// TIA Portal V20 export
FUNCTION_BLOCK "FB - TableCheck"   // FB3, LAD
TITLE = Equipment - TableCheck
{ S7_Optimized_Access := 'TRUE' }
// This function block contains all logic for controlling a TableCheck module.
// -This module consists of a table, a jig presense sensor and Indication lamp Red (NG) and green (Ok).
// 
// >> Block created by: Engr. Awais Ali
// >> Block creation date:  08-10-2025
// stored: MemoryReserve 100, SetENOAutomatically false
   VAR_INPUT
      i_xJigPresent : Bool;
   END_VAR
   VAR_OUTPUT
      q_xLampNG : Bool;
      q_xLampOK : Bool;
   END_VAR
   VAR_IN_OUT
      iq_tableCheck : "UDT-TableCheck";
      iq_Sabload_L : "UDT-SABload";
      iq_Sabload_R : "UDT-SABload";
      iq_Bas342 : "UDT-BAS342";
   END_VAR
   VAR
      iState : Int;
      OnDelay_JigL { S7_SetPoint := 'True'} : TON_TIME;
      OffDelay_JigL { S7_SetPoint := 'True'} : TOF_TIME;
      OnDelay_JigR { S7_SetPoint := 'True'} : TON_TIME;
      OffDelay_JigR { S7_SetPoint := 'True'} : TOF_TIME;
   END_VAR
BEGIN

REGION Network 1: control - left jig
   // Detect the presence of left side Jig.
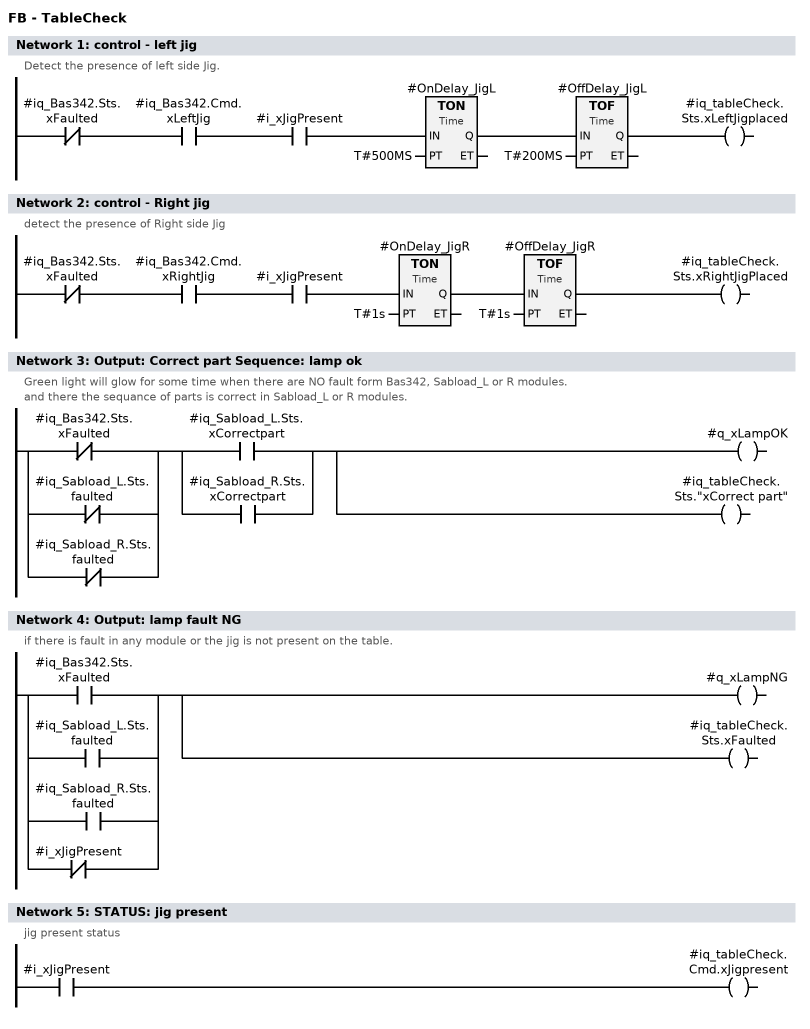
   RUNG wire#powerrail
      I_Contact( #iq_Bas342.Sts.xFaulted )
      Contact( #iq_Bas342.Cmd.xLeftJig )
      Contact( #i_xJigPresent )
      { S7_Templates := "time_type := Time" } #OnDelay_JigL.TON(pt := T#500MS, et =>)
      { S7_Templates := "time_type := Time" } #OffDelay_JigL.TOF(pt := T#200MS, et =>)
      Coil( #iq_tableCheck.Sts.xLeftJigplaced )
   END_RUNG
   // the same network as SCL:
   #OnDelay_JigL(IN := NOT #iq_Bas342.Sts.xFaulted AND #iq_Bas342.Cmd.xLeftJig AND #i_xJigPresent,   // TON
                 PT := T#500MS);
   #OffDelay_JigL(IN := #OnDelay_JigL.Q, PT := T#200MS);   // TOF
   #iq_tableCheck.Sts.xLeftJigplaced := #OffDelay_JigL.Q;
END_REGION

REGION Network 2: control - Right jig
   // detect the presence of Right side Jig
   RUNG wire#powerrail
      I_Contact( #iq_Bas342.Sts.xFaulted )
      Contact( #iq_Bas342.Cmd.xRightJig )
      Contact( #i_xJigPresent )
      { S7_Templates := "time_type := Time" } #OnDelay_JigR.TON(pt := T#1s, et =>)
      { S7_Templates := "time_type := Time" } #OffDelay_JigR.TOF(pt := T#1s, et =>)
      Coil( #iq_tableCheck.Sts.xRightJigPlaced )
   END_RUNG
   // the same network as SCL:
   #OnDelay_JigR(IN := NOT #iq_Bas342.Sts.xFaulted AND #iq_Bas342.Cmd.xRightJig AND #i_xJigPresent, PT := T#1s);   // TON
   #OffDelay_JigR(IN := #OnDelay_JigR.Q, PT := T#1s);   // TOF
   #iq_tableCheck.Sts.xRightJigPlaced := #OffDelay_JigR.Q;
END_REGION

REGION Network 3: Output: Correct part Sequence: lamp ok
   // Green light will glow for some time when there are NO fault form Bas342, Sabload_L or R modules. 
   // 
   // and there the sequance of parts is correct in Sabload_L or R modules.
   RUNG wire#powerrail
      I_Contact( #iq_Bas342.Sts.xFaulted )
      wire#w1
      Contact( #iq_Sabload_L.Sts.xCorrectpart )
      wire#w2
      Coil( #q_xLampOK )
   END_RUNG
   RUNG wire#powerrail
      I_Contact( #iq_Sabload_L.Sts.faulted )
   END_RUNG wire#w1
   RUNG wire#powerrail
      I_Contact( #iq_Sabload_R.Sts.faulted )
   END_RUNG wire#w1
   RUNG wire#w1
      Contact( #iq_Sabload_R.Sts.xCorrectpart )
   END_RUNG wire#w2
   RUNG wire#w2
      Coil( #iq_tableCheck.Sts."xCorrect part" )
   END_RUNG
   // the same network as SCL:
   #q_xLampOK := (NOT #iq_Bas342.Sts.xFaulted OR NOT #iq_Sabload_L.Sts.faulted OR NOT #iq_Sabload_R.Sts.faulted) AND (#iq_Sabload_L.Sts.xCorrectpart OR #iq_Sabload_R.Sts.xCorrectpart);
   #iq_tableCheck.Sts."xCorrect part" := #q_xLampOK;
END_REGION

REGION Network 4: Output: lamp fault NG
   // if there is fault in any module or the jig is not present on the table.
   RUNG wire#powerrail
      Contact( #iq_Bas342.Sts.xFaulted )
      wire#w1
      Coil( #q_xLampNG )
   END_RUNG
   RUNG wire#powerrail
      Contact( #iq_Sabload_L.Sts.faulted )
   END_RUNG wire#w1
   RUNG wire#powerrail
      Contact( #iq_Sabload_R.Sts.faulted )
   END_RUNG wire#w1
   RUNG wire#powerrail
      I_Contact( #i_xJigPresent )
   END_RUNG wire#w1
   RUNG wire#w1
      Coil( #iq_tableCheck.Sts.xFaulted )
   END_RUNG
   // the same network as SCL:
   #q_xLampNG := #iq_Bas342.Sts.xFaulted OR #iq_Sabload_L.Sts.faulted OR #iq_Sabload_R.Sts.faulted OR NOT #i_xJigPresent;
   #iq_tableCheck.Sts.xFaulted := #q_xLampNG;
END_REGION

REGION Network 5: STATUS: jig present
   // jig present status
   RUNG wire#powerrail
      Contact( #i_xJigPresent )
      Coil( #iq_tableCheck.Cmd.xJigpresent )
   END_RUNG
   // the same network as SCL:
   #iq_tableCheck.Cmd.xJigpresent := #i_xJigPresent;
END_REGION
END_FUNCTION_BLOCK
